FUNCTION_BLOCK fbServo
VAR_INPUT
	Interlock_1 : BOOL;
	Interlock_2 : BOOL;
	Interlock_3 : BOOL;
	Interlock_4 : BOOL;
	Interlock_5 : BOOL;
	Interlock_6 : BOOL;
	Interlock_7 : BOOL;

	AutoGoToPos : BOOL;
	Stop : BOOL;
	AutoPosSp : REAL;
	AutoSpeedSp : REAL; // % from max
	AutoAccSp : REAL; // % from max
	AutoJerkSp : REAL; // % from max
END_VAR
VAR_OUTPUT
	AutoMan : BOOL;
	PositionReached : BOOL;
	Running : BOOL;
	Faulted : BOOL;

	Position : REAL;
	Speed : REAL;
END_VAR
VAR
	Interlock_OK : BOOL;
	AutoReq : BOOL;
	ManReq : BOOL;

	ManPosSP : REAL;
	ManSpeedSP : REAL;
	ManAccSP : REAL;
	ManJerk : REAL;
	GoToPosition : BOOL;
	HomeReq : BOOL;
	JogForward : BOOL;
	JogBackward : BOOL;
	ClearFault : BOOL;
	FaultID : BOOL;
	
	PosSP : REAL;
	SpeedSP : REAL;
	AccSP : REAL;
	JerkSP : REAL;

	strInterlock_1 : STRING;
	strInterlock_2 : STRING;
	strInterlock_3 : STRING;
	strInterlock_4 : STRING;
	strInterlock_5 : STRING;
	strInterlock_6 : STRING;
	strInterlock_7 : STRING;
	strAutoMan : STRING;
END_VAR
VAR // added by the converter: edge detectors and wires of the graphical bodies
    _w1, _w2, _w3, _w4, _w5, _w6, _w7, _w8 : BOOL;
END_VAR

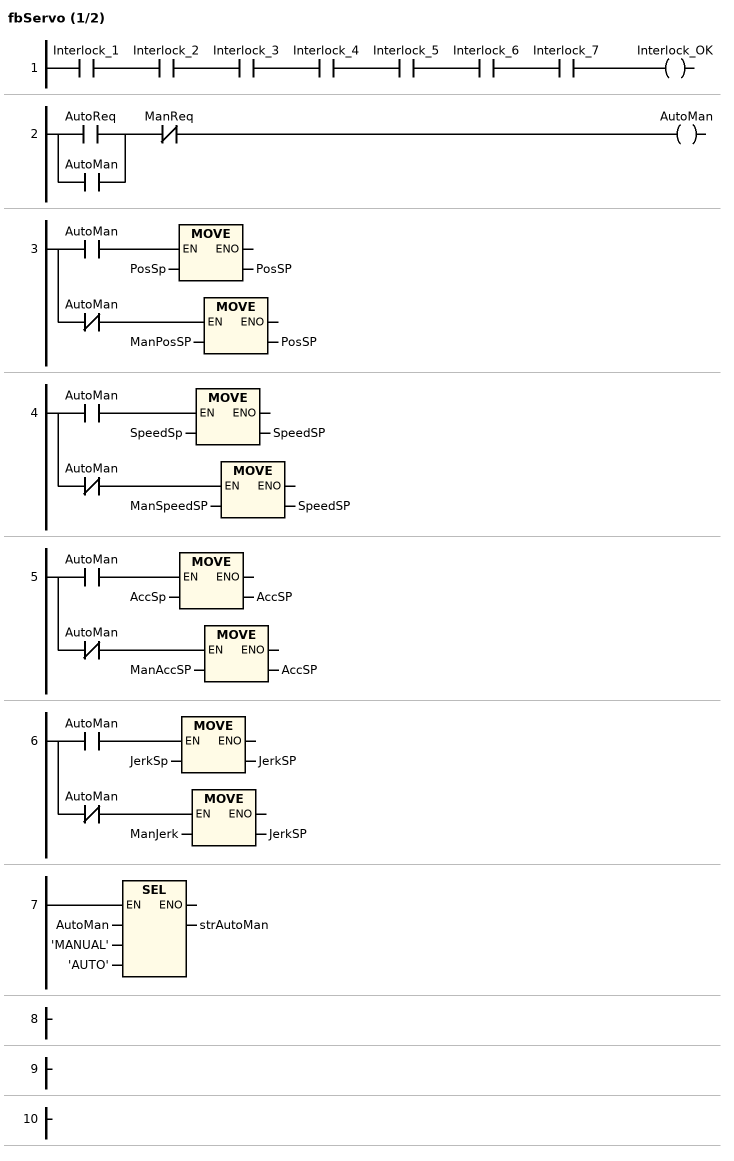
// NETWORK 1
Interlock_OK := Interlock_1 AND Interlock_2 AND Interlock_3 AND Interlock_4 AND Interlock_5 AND Interlock_6 AND Interlock_7;

// NETWORK 2
AutoMan := (AutoReq OR AutoMan) AND NOT ManReq;

// NETWORK 3
_w1 := AutoMan;
IF _w1 THEN PosSP := PosSp; END_IF
_w2 := NOT AutoMan;
IF _w2 THEN PosSP := ManPosSP; END_IF
(* _w1 OR _w2; result not used *)

// NETWORK 4
_w3 := AutoMan;
IF _w3 THEN SpeedSP := SpeedSp; END_IF
_w4 := NOT AutoMan;
IF _w4 THEN SpeedSP := ManSpeedSP; END_IF
(* _w3 OR _w4; result not used *)

// NETWORK 5
_w5 := AutoMan;
IF _w5 THEN AccSP := AccSp; END_IF
_w6 := NOT AutoMan;
IF _w6 THEN AccSP := ManAccSP; END_IF
(* _w5 OR _w6; result not used *)

// NETWORK 6
_w7 := AutoMan;
IF _w7 THEN JerkSP := JerkSp; END_IF
_w8 := NOT AutoMan;
IF _w8 THEN JerkSP := ManJerk; END_IF
(* _w7 OR _w8; result not used *)

// NETWORK 7
strAutoMan := SEL(AutoMan, 'MANUAL', 'AUTO');

// NETWORK 8

// NETWORK 9

// NETWORK 10

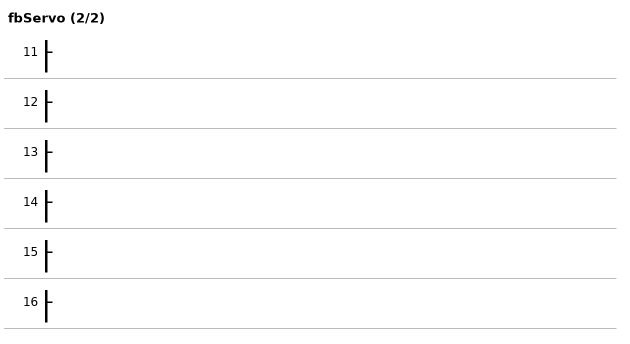
// NETWORK 11

// NETWORK 12

// NETWORK 13

// NETWORK 14

// NETWORK 15

// NETWORK 16

END_FUNCTION_BLOCK

(* stored: Version 1.1.0.1, ProductVersion 3.1.4022.17
   POU fbServo: Id {06f35ab6-0b69-4919-8f62-c873445ba8c3}, SpecialFunc None *)
